PROGRAM MAIN
VAR
	fActualValue : REAL;
	fTargetValue : REAL := 50.0 ;
	fTolerance : REAL := 2.0 ;
	
	bTargetReached : BOOL;
END_VAR

IF (fActualValue >= (fTargetValue - fTolerance)) AND (FaCTUALvALUE <= (fTargetValue + fTolerance)) THEN
	bTargetReached := TRUE;
ELSE
	bTargetReached := FALSE;
END_IF

END_PROGRAM

(* stored: Version 1.1.0.1
   POU MAIN: Id {329ee81f-6c4b-411e-8d0f-ec979ee02565}, SpecialFunc None *)
